INTERFACE I_Motor

PROPERTY CurrentPosition : REAL
GET
END_GET
END_PROPERTY

PROPERTY CurrentSpeed : real
GET
END_GET
END_PROPERTY

METHOD Jog
VAR_INPUT
END_VAR
END_METHOD

PROPERTY LimitPositionForward : real
GET
END_GET
SET
END_SET
END_PROPERTY

PROPERTY LimitPositionReverse : real
GET
END_GET
SET
END_SET
END_PROPERTY

METHOD MoveAbsolute
VAR_INPUT
END_VAR
END_METHOD

METHOD MoveRelative
VAR_INPUT
END_VAR
END_METHOD

METHOD PowerOn
VAR_INPUT
END_VAR
END_METHOD

METHOD Reset
VAR_INPUT
END_VAR
END_METHOD

PROPERTY SetPosition : REAL
GET
END_GET
SET
END_SET
END_PROPERTY

PROPERTY SetSpeed : REAL
GET
END_GET
SET
END_SET
END_PROPERTY

METHOD Stop
END_METHOD

END_INTERFACE

(* stored: Version 1.1.0.1, ProductVersion 3.1.4026.18
   Itf I_Motor: Id {0f878f3d-e223-42ff-9cbd-c4403f98b8fe}
   Property CurrentPosition: Id {e701f28c-3131-41d7-a7d8-b744ca2b041d}
   Get Get: Id {6192cb32-65aa-45fa-9e6a-fe2286ddc8a2}
   Property CurrentSpeed: Id {e0330a7a-01f0-4cc3-9c0d-6e092b3f19a8}
   Get Get: Id {97663ae7-ab4f-4e5c-a7d9-b68d72004717}
   Method Jog: Id {d39e881a-21f4-4b05-8f60-7c1b98288ca2}
   Property LimitPositionForward: Id {fff801f1-a6fe-4d2a-9541-27dcd11a56d1}
   Get Get: Id {766ec37e-da86-4881-9d25-76ac1c3d0d69}
   Set Set: Id {0a67063e-b33b-4676-884a-128b9ba46f8b}
   Property LimitPositionReverse: Id {29dddabf-6a49-497e-9cb2-ff1a2e240d7f}
   Get Get: Id {73b85b3a-d3d6-4c1a-b5c2-acf48a67fa7e}
   Set Set: Id {fa884763-6220-4b94-96fc-8a9afa22e2e0}
   Method MoveAbsolute: Id {bb6dcfc0-b16f-4d80-bdef-a1273a2a3a70}
   Method MoveRelative: Id {1478f5ea-bc89-4224-b4bd-ea2485cdf0ab}
   Method PowerOn: Id {87af280f-7bab-4f1b-82cf-30a988f1a544}
   Method Reset: Id {8785d36c-8c85-4d61-9883-7664b97f1338}
   Property SetPosition: Id {1852035f-54da-4bee-92b7-8aee4a7be76d}
   Get Get: Id {4a4c288d-2f80-4f22-8db9-a63f00fa011e}
   Set Set: Id {d5b4f39a-2dcd-44a6-80f9-70af36a1ce01}
   Property SetSpeed: Id {9b0b9027-20e1-4cb2-bb54-f155330a9f95}
   Get Get: Id {8661cc88-961a-4120-9c0a-3970e7a963f2}
   Set Set: Id {ed6e81b4-95ad-49e4-870a-16b1d2e7a692}
   Method Stop: Id {1e0fac7f-07d9-40d3-9a49-88f4ee562921} *)
